// TwinCAT 3 PLC project ConveyorsExtSet
// ProgramVersion: 3.1.4023.0
// libraries:
//   Tc2_Standard, * (Beckhoff Automation GmbH)
//   Tc2_System, * (Beckhoff Automation GmbH)
//   Tc3_Module, * (Beckhoff Automation GmbH)
// project tree:
//   DUTs/ ConveyorLSC.TcPOU (not stored), ConveyorMode.TcDUT (not stored), ConveyorSC.TcPOU
//   / PlcTask.TcTTO
//   POUs/ MAIN.TcPOU
// (motion and I/O tree: see PLC project drivesv1)
// real-time tasks:
//   TASK PlcTask: cycle T#10ms, priority 20, ADS port 350
//   TASK PlcTask1: cycle T#10ms, priority 21, ADS port 351
//   TASK PlcTask2: cycle T#10ms, priority 22, ADS port 352
//   TASK PlcTask3: cycle T#10ms, priority 23, ADS port 353
//   TASK PlcTask4: cycle T#10ms, priority 24, ADS port 354

CONFIGURATION ConveyorsExtSet
    RESOURCE PLC ON TwinCAT3
        TASK PlcTask(INTERVAL := T#10ms, PRIORITY := 24);
        PROGRAM MAIN WITH PlcTask : MAIN;
    END_RESOURCE
END_CONFIGURATION

// ---- POUs/MAIN.TcPOU
PROGRAM MAIN
VAR
	sc1 : ConveyorSC;
	sc2 : ConveyorSC;
	sc3 : ConveyorSC;
	sc4 : ConveyorSC;
	lsc5 : ConveyorLSC;
	lsc6 : ConveyorLSC;
	lsc7 : ConveyorLSC;
	lsc8 : ConveyorLSC;
	
END_VAR
VAR
	arr : ARRAY[1..8] OF POINTER TO ConveyorSC;
	i : INT;
	j : INT;
	
	linkStart : INT := -1;
	linkEnd : INT := -1;
	chainMode : ConveyorMode;
END_VAR
(*
in this module, conveyors are implemented as a linked list
each conveyor's mode is determined by the actual mode (not requested mode) of its adjacent conveyors
*)

//double click on these for online write
(*
conveyor linking algorithm:
	-find a chain where all conveyors are occupied
	-find highest priority request between the chain
	-set the actual mode all conveyors in the chain to that highest priority request
*)

call();

sc1.trueMode;
sc2.trueMode;
sc3.trueMode;
sc4.trueMode;
lsc5.trueMode;
lsc6.trueMode;
lsc7.trueMode;
lsc8.trueMode;

sc1.requestedMode;
sc2.requestedMode;
sc3.requestedMode;
sc4.requestedMode;
lsc5.requestedMode;
lsc6.requestedMode;
lsc7.requestedMode;
lsc8.requestedMode;


linkStart := -1;
linkEnd := -1;
chainMode := 0;

FOR i:=1 TO 8 BY 1 DO
	
	IF arr[i]^.IsOccupied THEN
		IF linkStart = -1 THEN
			linkStart := i;
		END_IF
		
		chainMode := MAX(chainMode, arr[i]^.requestedMode);
		linkEnd := i;
	
	ELSIF linkStart <> -1 AND linkEnd <> -1 THEN //set all conveyor operations to priorityInLink
		
		FOR j:=linkStart TO linkEnd BY 1 DO
			arr[j]^.setMode(chainMode);
		END_FOR
		
		linkStart := -1;
		linkEnd := -1;
		
		chainMode := ConveyorMode.IDLE;
		arr[i]^.setMode(ConveyorMode.IDLE);
		
		CONTINUE;
	END_IF
	
END_FOR

IF linkStart > -1 AND linkEnd > -1 THEN
	FOR j:=linkStart TO linkEnd BY 1 DO
		arr[j]^.setMode(chainMode);
	END_FOR
END_IF




call();

ACTION call:
arr[1] := ADR(sc1);
arr[2] := ADR(sc2);
arr[3] := ADR(sc3);
arr[4] := ADR(sc4);
arr[5] := ADR(lsc5);
arr[6] := ADR(lsc6);
arr[7] := ADR(lsc7);
arr[8] := ADR(lsc8);

FOR i:=1 TO 8-1 BY 1 DO
	
	arr[i]^.join(arr[i+1]);
	
END_FOR


sc1(error=> , position=> , velocity=> );
sc2(error=> , position=> , velocity=> );
sc3(error=> , position=> , velocity=> );
sc4(error=> , position=> , velocity=> );

lsc5(
	error=> , 
	position=> , 
	velocity=> , 
	lifterError=> , 
	extended=> , 
	retracted=> );
	
lsc6(
	error=> , 
	position=> , 
	velocity=> , 
	lifterError=> , 
	extended=> , 
	retracted=> );
	
lsc7(
	error=> , 
	position=> , 
	velocity=> , 
	lifterError=> , 
	extended=> , 
	retracted=> );
	
lsc8(
	error=> , 
	position=> , 
	velocity=> , 
	lifterError=> , 
	extended=> , 
	retracted=> );
END_ACTION

END_PROGRAM

// ---- DUTs/ConveyorSC.TcPOU
FUNCTION_BLOCK ConveyorSC
VAR_OUTPUT
	trueMode : ConveyorMode;
	requestedMode : ConveyorMode;
	
	error AT %I* : BOOL;
	position AT %I* : REAL;
	velocity AT %I* : REAL;
END_VAR
VAR
	enable AT %Q* : BOOL := TRUE;
	direction AT %Q* : BOOL; //FALSE = forward, TRUE = backward
	pulse AT %Q* : BOOL;
	reset AT %Q* : BOOL;
	
	sensorEntry AT %I* : BOOL := TRUE;
	sensorExit AT %I* : BOOL;
END_VAR
VAR
	//nextConveyor : POINTER TO ConveyorSC;
	//prevConveyor : POINTER TO ConveyorSC;
	
	pulser : TP; //pulses are assumed to be low-high-low
END_VAR
VAR_STAT CONSTANT
	pulseWidth : TIME := T#50MS;
END_VAR

override();

sequence();

METHOD backward : BOOL
VAR_INPUT
END_VAR
END_METHOD

METHOD forward : BOOL
VAR_INPUT
END_VAR
END_METHOD

{attribute 'monitoring' := 'call'}
PROPERTY IsOccupied : BOOL
GET
IsOccupied := sensorExit OR sensorEntry;
END_GET
END_PROPERTY

METHOD join : BOOL
VAR_INPUT
	conveyor : POINTER TO ConveyorSC;
END_VAR
//nextConveyor := conveyor;
//conveyor^.prevConveyor := THIS;
END_METHOD

METHOD PROTECTED override : BOOL
VAR_INPUT
END_VAR
END_METHOD

METHOD reset : BOOL
VAR_INPUT
END_VAR
position := 0;
velocity := velocity; //no change
END_METHOD

METHOD PROTECTED sequence : BOOL
VAR_INPUT
END_VAR
direction := (trueMode = ConveyorMode.BACKWARD); //set direction bit

pulser(IN:= , PT:= pulseWidth, Q=> pulse, ET=> );
pulser.IN := 
	enable AND 
	NOT error AND 
	NOT reset AND 
	(trueMode = ConveyorMode.FORWARD OR trueMode = ConveyorMode.BACKWARD)
	AND pulser.Q; //ends pulse itself
END_METHOD

METHOD setMode : BOOL
VAR_INPUT
	mode : ConveyorMode;
END_VAR
trueMode := mode;
END_METHOD

METHOD target : BOOL
VAR_INPUT
	targetPosition : REAL;
END_VAR
END_METHOD

END_FUNCTION_BLOCK
